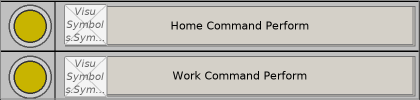
VISUALIZATION vActuator_Frame  // 420x100
VAR_INPUT
	iTextIndex1 : INT;
	iTextIndex2 : INT;
END_VAR
VAR_IN_OUT
	fbActuator:FB_ActuatorOOP_TC;
END_VAR
    Rectangle (0,51 420x50)
    Rectangle (0,1 420x50)
    Rectangle (0,1 55x100)
    Button (65,6 350x40), "Home Command Perform", pressed state: fbActuator.bHomeCmd, input disabled if: NOT fbActuator.bManualMode, text list: 'ActuatorNames', text index: iTextIndex1
        OnMouseClick: execute { fbActuator.mGoToHome(TRUE); }
    Button (65,56 350x40), "Work Command Perform", pressed state: fbActuator.bWorkCmd, input disabled if: NOT fbActuator.bManualMode, text list: 'ActuatorNames', text index: iTextIndex2
        OnMouseClick: execute { fbActuator.mGoToWork(TRUE); }
    Lamp1 (5,52 50x50), variable: fbActuator.fbTON_WorkPositionDelayed.Q, style: Lamp-Lamp1-Yellow
    Lamp1 (5,1 50x50), variable: fbActuator.fbTON_HomePositionDelayed.Q, style: Lamp-Lamp1-Yellow
    Image (64,56 43x41), invisible if: fbActuator.pAllowWork, image: VisuSymbols.Symbols.Lock
    Image (64,4 43x41), invisible if: fbActuator.pAllowHome, image: VisuSymbols.Symbols.Lock
END_VISUALIZATION

(* stored: Version 1.1.0.1, ProductVersion 3.1.4024.15
   Visu vActuator_Frame: Id {a49e921c-8a0f-4cf3-8dff-74d4448b6a24} *)
